Staubli VAL3: Txt_initData.pgx

program Txt_initData()
  local num l_nInit
begin
  while size(sString)>1
    $ddel(sString,size(sString)-1)
  endWhile
  while size(pfrmCad)>1
    $ddel(pfrmCad,size(pfrmCad)-1)
  endWhile
  while size(nPulse)>1
    $ddel(nPulse,size(nPulse)-1)
  endWhile
  pfrmCad[0].trsf={0,0,0,0,0,0}
  sString[0]=""
  nPulse[0]=0
  for l_nInit=1 to 1499
    $dins(sString,l_nInit)
    $dins(pfrmCad,l_nInit)
    $dins(nPulse,l_nInit)
  endFor
  bTxtPrSv=false
  sScrPts="NotReady"
  call hmi_refreshmain()


end
